TYPE Struct_M_lakeshore :
STRUCT
	Temperature:LREAL;(*Celsius*)
	Resistance:LREAL;
END_STRUCT
END_TYPE

(* stored: Version 1.1.0.1, ProductVersion 3.1.4024.6
   DUT Struct_M_lakeshore: Id {c89bef22-063c-4729-ae7c-eeb6c5f9a7b4} *)
